FUNCTION alg_a_zdown : BOOL
VAR_INPUT
	state: STATE;
END_VAR

alg_a_zdown := state.dvar_M_example_controller_a_zdown;

END_FUNCTION

(* stored: Version 1.1.0.1, ProductVersion 3.1.4022.18
   POU alg_a_zdown: Id {3b732896-524e-4f57-8238-fe4577818d0f}, SpecialFunc None *)
